Yaskawa INFORM job: sMulti_Axis_right_toolchange.JBI

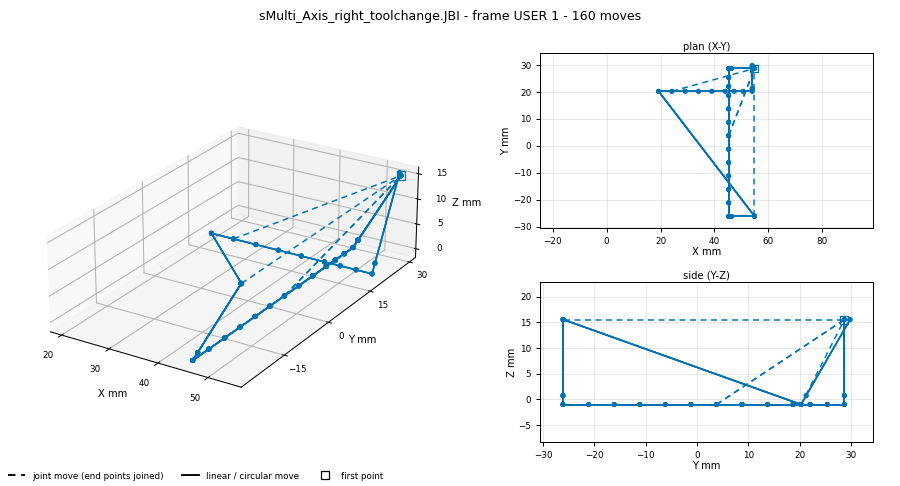
[picture p0: tool path of sMulti_Axis_right_toolchange.JBI in frame USER 1, 160 of 160 moves have a stored position in this frame; points joined in program order, loops and branches not executed]
/JOB
//NAME sMulti_Axis_right_toolchange
//POS
///NPOS 17,0,0,0,0,0
///USER 1
///TOOL 2
///POSTYPE USER
///RECTAN
///RCONF 1,0,0,0,0,0
C00000=50.999,-29.823,15.536,-90.000,-150.794,-116.565
C00001=50.999,-21.274,0.729,-90.000,-150.794,-116.565
C00002=50.999,-20.274,-1.003,-90.000,-150.794,-116.565
C00003=47.666,-20.274,-1.003,-90.000,-150.794,-116.565
C00004=44.332,-20.274,-1.003,-90.000,-150.794,-116.565
C00005=40.999,-20.274,-1.003,-90.000,-150.794,-116.565
C00006=36.223,-20.274,-1.003,-90.000,-150.794,-116.565
C00007=31.447,-20.274,-1.003,-90.000,-150.794,-116.565
C00008=26.671,-20.274,-1.003,-90.000,-150.794,-116.565
C00009=21.896,-20.274,-1.003,-90.000,-150.794,-116.565
C00010=17.120,-20.274,-1.003,-90.000,-150.794,-116.565
C00011=12.344,-20.274,-1.003,-90.000,-150.794,-116.565
C00012=7.568,-20.274,-1.003,-90.000,-150.794,-116.565
C00013=2.792,-20.274,-1.003,-90.000,-150.794,-116.565
C00014=-1.983,-20.274,-1.003,-90.000,-150.794,-116.565
C00015=-6.759,-20.274,-1.003,-90.000,-150.794,-116.565
C00016=-11.535,-20.274,-1.003,-90.000,-150.794,-116.565
C00017=-16.311,-20.274,-1.003,-90.000,-150.794,-116.565
C00018=-21.087,-20.274,-1.003,-90.000,-150.794,-116.565
C00019=-25.862,-20.274,-1.003,-90.000,-150.794,-116.565
C00020=-30.638,-20.274,-1.003,-90.000,-150.794,-116.565
C00021=-35.414,-20.274,-1.003,-90.000,-150.794,-116.565
C00022=-40.190,-20.274,-1.003,-90.000,-150.794,-116.565
C00023=-44.966,-20.274,-1.003,-90.000,-150.794,-116.565
C00024=-48.299,-20.274,-1.003,-90.000,-150.794,-116.565
C00025=-51.632,-20.274,-1.003,-90.000,-150.794,-116.565
C00026=-54.966,-20.274,-1.003,-90.000,-150.794,-116.565
C00027=-54.966,-21.274,0.729,-90.000,-150.794,-116.565
C00028=-54.966,-29.823,15.536,-90.000,-150.794,-116.565
C00000=53.984,-29.817,15.539,-90.000,-150.794,-116.565
C00001=53.984,-24.817,6.879,-90.000,-150.794,-116.565
C00002=53.984,-20.744,-0.175,-90.000,-150.794,-116.565
C00003=53.705,-20.407,-0.758,-90.000,-150.794,-116.565
C00004=53.031,-20.268,-1.000,-90.000,-150.794,-116.565
C00005=-55.536,-20.268,-1.000,-90.000,-150.794,-116.565
C00006=-56.209,-20.407,-0.758,-90.000,-150.794,-116.565
C00007=-56.488,-20.744,-0.175,-90.000,-150.794,-116.565
C00008=-56.488,-29.817,15.539,-90.000,-150.794,-116.565
C00000=-54.823,-30.003,15.536,180.000,-152.507,146.310
C00001=-46.274,-30.003,0.729,180.000,-152.507,146.310
C00002=-45.274,-30.003,-1.003,180.000,-152.507,146.310
C00003=-45.274,-26.669,-1.003,180.000,-152.507,146.310
C00004=-45.274,-23.336,-1.003,180.000,-152.507,146.310
C00005=-45.274,-20.003,-1.003,180.000,-152.507,146.310
C00006=-45.274,-15.558,-1.003,180.000,-152.507,146.310
C00007=-45.274,-11.113,-1.003,180.000,-152.507,146.310
C00008=-45.274,-6.668,-1.003,180.000,-152.507,146.310
C00009=-45.274,-2.223,-1.003,180.000,-152.507,146.310
C00010=-45.274,2.223,-1.003,180.000,-152.507,146.310
C00011=-45.274,6.668,-1.003,180.000,-152.507,146.310
C00012=-45.274,11.113,-1.003,180.000,-152.507,146.310
C00013=-45.274,15.558,-1.003,180.000,-152.507,146.310
C00014=-45.274,20.003,-1.003,-180.000,-152.507,146.310
C00015=-45.274,23.336,-1.003,-180.000,-152.507,146.310
C00016=-45.274,26.669,-1.003,-180.000,-152.507,146.310
C00017=-45.274,30.003,-1.003,-180.000,-152.507,146.310
C00018=-46.274,30.003,0.729,-180.000,-152.507,146.310
C00019=-54.823,30.003,15.536,-180.000,-152.507,146.310
C00000=54.301,-29.817,15.539,-90.000,-150.794,-116.565
C00001=54.301,-24.817,6.879,-90.000,-150.794,-116.565
C00002=54.301,-20.903,0.100,-90.000,-150.794,-116.565
C00003=53.929,-20.454,-0.678,-90.000,-150.794,-116.565
C00004=53.031,-20.268,-1.000,-90.000,-150.794,-116.565
C00005=-55.536,-20.268,-1.000,-90.000,-150.794,-116.565
C00006=-56.434,-20.454,-0.678,-90.000,-150.794,-116.565
C00007=-56.806,-20.903,0.100,-90.000,-150.794,-116.565
C00008=-56.806,-29.817,15.539,-90.000,-150.794,-116.565
C00000=-54.969,29.823,15.536,90.000,-150.794,63.435
C00001=-54.969,21.274,0.729,90.000,-150.794,63.435
C00002=-54.969,20.274,-1.003,90.000,-150.794,63.435
C00003=-51.636,20.274,-1.003,90.000,-150.794,63.435
C00004=-48.303,20.274,-1.003,90.000,-150.794,63.435
C00005=-44.969,20.274,-1.003,90.000,-150.794,63.435
C00006=-40.029,20.274,-1.003,90.000,-150.794,63.435
C00007=-35.088,20.274,-1.003,90.000,-150.794,63.435
C00008=-30.147,20.274,-1.003,90.000,-150.794,63.435
C00009=-25.206,20.274,-1.003,90.000,-150.794,63.435
C00010=-20.266,20.274,-1.003,90.000,-150.794,63.435
C00011=-15.325,20.274,-1.003,90.000,-150.794,63.435
C00012=-10.384,20.274,-1.003,90.000,-150.794,63.435
C00013=-5.443,20.274,-1.003,90.000,-150.794,63.435
C00014=-0.502,20.274,-1.003,90.000,-150.794,63.435
C00015=4.438,20.274,-1.003,90.000,-150.794,63.435
C00016=9.379,20.274,-1.003,90.000,-150.794,63.435
C00017=14.320,20.274,-1.003,90.000,-150.794,63.435
C00018=19.261,20.274,-1.003,90.000,-150.794,63.435
C00019=24.201,20.274,-1.003,90.000,-150.794,63.435
C00020=29.142,20.274,-1.003,90.000,-150.794,63.435
C00021=34.083,20.274,-1.003,90.000,-150.794,63.435
C00022=39.024,20.274,-1.003,90.000,-150.794,63.435
C00023=43.965,20.274,-1.003,90.000,-150.794,63.435
C00024=47.298,20.274,-1.003,90.000,-150.794,63.435
C00025=50.631,20.274,-1.003,90.000,-150.794,63.435
C00026=53.965,20.274,-1.003,90.000,-150.794,63.435
C00027=53.965,21.274,0.729,90.000,-150.794,63.435
C00028=53.965,29.823,15.536,90.000,-150.794,63.435
C00000=-54.969,29.823,15.536,90.000,-150.794,63.435
C00001=-54.969,21.274,0.729,90.000,-150.794,63.435
C00002=-54.969,20.274,-1.003,90.000,-150.794,63.435
C00003=-51.636,20.274,-1.003,90.000,-150.794,63.435
C00004=-48.303,20.274,-1.003,90.000,-150.794,63.435
C00005=-44.969,20.274,-1.003,90.000,-150.794,63.435
C00006=-40.029,20.274,-1.003,90.000,-150.794,63.435
C00007=-35.088,20.274,-1.003,90.000,-150.794,63.435
C00008=-30.147,20.274,-1.003,90.000,-150.794,63.435
C00009=-25.206,20.274,-1.003,90.000,-150.794,63.435
C00010=-20.266,20.274,-1.003,90.000,-150.794,63.435
C00011=-15.325,20.274,-1.003,90.000,-150.794,63.435
C00012=-10.384,20.274,-1.003,90.000,-150.794,63.435
C00013=-5.443,20.274,-1.003,90.000,-150.794,63.435
C00014=-0.502,20.274,-1.003,90.000,-150.794,63.435
C00015=4.438,20.274,-1.003,90.000,-150.794,63.435
C00016=9.379,20.274,-1.003,90.000,-150.794,63.435
C00017=14.320,20.274,-1.003,90.000,-150.794,63.435
C00018=19.261,20.274,-1.003,90.000,-150.794,63.435
C00019=24.201,20.274,-1.003,90.000,-150.794,63.435
C00020=29.142,20.274,-1.003,90.000,-150.794,63.435
C00021=34.083,20.274,-1.003,90.000,-150.794,63.435
C00022=39.024,20.274,-1.003,90.000,-150.794,63.435
C00023=43.965,20.274,-1.003,90.000,-150.794,63.435
C00024=47.298,20.274,-1.003,90.000,-150.794,63.435
C00025=50.631,20.274,-1.003,90.000,-150.794,63.435
C00026=53.965,20.274,-1.003,90.000,-150.794,63.435
C00027=53.965,21.274,0.729,90.000,-150.794,63.435
C00028=53.965,29.823,15.536,90.000,-150.794,63.435
C00000=54.817,28.503,15.539,0.000,-152.507,-33.690
C00001=46.268,28.503,0.732,0.000,-152.507,-33.690
C00002=45.268,28.503,-1.000,0.000,-152.507,-33.690
C00003=45.268,25.169,-1.000,0.000,-152.507,-33.690
C00004=45.268,21.836,-1.000,0.000,-152.507,-33.690
C00005=45.268,18.503,-1.000,0.000,-152.507,-33.690
C00006=45.268,13.573,-1.000,0.000,-152.507,-33.690
C00007=45.268,8.644,-1.000,0.000,-152.507,-33.690
C00008=45.268,3.715,-1.000,0.000,-152.507,-33.690
C00009=45.268,-1.214,-1.000,0.000,-152.507,-33.690
C00010=45.268,-6.144,-1.000,0.000,-152.507,-33.690
C00011=45.268,-11.073,-1.000,0.000,-152.507,-33.690
C00012=45.268,-16.002,-1.000,0.000,-152.507,-33.690
C00013=45.268,-19.336,-1.000,0.000,-152.507,-33.690
C00014=45.268,-22.669,-1.000,0.000,-152.507,-33.690
C00015=45.268,-26.002,-1.000,0.000,-152.507,-33.690
C00016=46.268,-26.002,0.732,0.000,-152.507,-33.690
C00017=54.817,-26.002,15.539,0.000,-152.507,-33.690
C00000=54.817,28.728,15.539,0.000,-152.507,-33.690
C00001=46.268,28.728,0.732,0.000,-152.507,-33.690
C00002=45.268,28.728,-1.000,0.000,-152.507,-33.690
C00003=45.268,25.395,-1.000,0.000,-152.507,-33.690
C00004=45.268,22.062,-1.000,0.000,-152.507,-33.690
C00005=45.268,18.728,-1.000,0.000,-152.507,-33.690
C00006=45.268,13.751,-1.000,0.000,-152.507,-33.690
C00007=45.268,8.773,-1.000,0.000,-152.507,-33.690
C00008=45.268,3.795,-1.000,0.000,-152.507,-33.690
C00009=45.268,-1.182,-1.000,0.000,-152.507,-33.690
C00010=45.268,-6.160,-1.000,0.000,-152.507,-33.690
C00011=45.268,-11.138,-1.000,0.000,-152.507,-33.690
C00012=45.268,-16.115,-1.000,0.000,-152.507,-33.690
C00013=45.268,-21.115,-1.000,0.000,-152.507,-33.690
C00014=45.268,-26.115,-1.000,0.000,-152.507,-33.690
C00015=46.268,-26.115,0.732,0.000,-152.507,-33.690
C00016=54.817,-26.115,15.539,0.000,-152.507,-33.690
//INST
///ATTR SC,RW,RJ
////FRAME USER 1
///GROUP1 RB1
///LVARS 2,0,0,0,0,0,0,0
NOP
SET LB000 1
SET LB001 25
MOVJ C00000 VJ=17
MOVL C00001 V=17 PL=LB000 ACC=LB001 DEC=LB001
' Lead In Move Starts
MOVL C00002 V=17 PL=LB000 ACC=LB001 DEC=LB001
' Cutting Move Starts
MOVL C00003 V=17 PL=LB000 ACC=LB001 DEC=LB001
MOVL C00004 V=17 PL=LB000 ACC=LB001 DEC=LB001
MOVL C00005 V=17 PL=LB000 ACC=LB001 DEC=LB001
MOVL C00006 V=17 PL=LB000 ACC=LB001 DEC=LB001
MOVL C00007 V=17 PL=LB000 ACC=LB001 DEC=LB001
MOVL C00008 V=17 PL=LB000 ACC=LB001 DEC=LB001
MOVL C00009 V=17 PL=LB000 ACC=LB001 DEC=LB001
MOVL C00010 V=17 PL=LB000 ACC=LB001 DEC=LB001
MOVL C00011 V=17 PL=LB000 ACC=LB001 DEC=LB001
MOVL C00012 V=17 PL=LB000 ACC=LB001 DEC=LB001
MOVL C00013 V=17 PL=LB000 ACC=LB001 DEC=LB001
MOVL C00014 V=17 PL=LB000 ACC=LB001 DEC=LB001
MOVL C00015 V=17 PL=LB000 ACC=LB001 DEC=LB001
MOVL C00016 V=17 PL=LB000 ACC=LB001 DEC=LB001
MOVL C00017 V=17 PL=LB000 ACC=LB001 DEC=LB001
MOVL C00018 V=17 PL=LB000 ACC=LB001 DEC=LB001
MOVL C00019 V=17 PL=LB000 ACC=LB001 DEC=LB001
MOVL C00020 V=17 PL=LB000 ACC=LB001 DEC=LB001
MOVL C00021 V=17 PL=LB000 ACC=LB001 DEC=LB001
MOVL C00022 V=17 PL=LB000 ACC=LB001 DEC=LB001
MOVL C00023 V=17 PL=LB000 ACC=LB001 DEC=LB001
MOVL C00024 V=17 PL=LB000 ACC=LB001 DEC=LB001
MOVL C00025 V=17 PL=LB000 ACC=LB001 DEC=LB001
MOVL C00026 V=17 PL=LB000 ACC=LB001 DEC=LB001
' Lead Out Move Starts
MOVL C00027 V=17 PL=LB000 ACC=LB001 DEC=LB001
' Rapid Move Starts
MOVL C00028 V=17 PL=LB000 ACC=LB001 DEC=LB001
' By Autodesk Fusion CAM 2.0.20494
' Tool = 8
' Spindle = 6000 RPM
' Set Position Level
' Set Acceleration
' Program Start
' First Toolpath Point
' Last Toolpath Point
MOVJ C00000 VJ=17
MOVL C00001 V=17 PL=LB000 ACC=LB001 DEC=LB001
' Plunge Move Starts
MOVL C00002 V=8 PL=LB000 ACC=LB001 DEC=LB001
' Lead In Move Starts
MOVL C00003 V=17 PL=LB000 ACC=LB001 DEC=LB001
MOVL C00004 V=17 PL=LB000 ACC=LB001 DEC=LB001
' Cutting Move Starts
MOVL C00005 V=17 PL=LB000 ACC=LB001 DEC=LB001
' Lead Out Move Starts
MOVL C00006 V=17 PL=LB000 ACC=LB001 DEC=LB001
MOVL C00007 V=17 PL=LB000 ACC=LB001 DEC=LB001
' Rapid Move Starts
MOVL C00008 V=17 PL=LB000 ACC=LB001 DEC=LB001
' By Autodesk Fusion CAM 2.0.20494
' Tool = 2
' Spindle = 5000 RPM
' Set Position Level
' Set Acceleration
' Program Start
' First Toolpath Point
' Last Toolpath Point
MOVJ C00000 VJ=17
MOVL C00001 V=17 PL=LB000 ACC=LB001 DEC=LB001
' Lead In Move Starts
MOVL C00002 V=17 PL=LB000 ACC=LB001 DEC=LB001
' Cutting Move Starts
MOVL C00003 V=17 PL=LB000 ACC=LB001 DEC=LB001
MOVL C00004 V=17 PL=LB000 ACC=LB001 DEC=LB001
MOVL C00005 V=17 PL=LB000 ACC=LB001 DEC=LB001
MOVL C00006 V=17 PL=LB000 ACC=LB001 DEC=LB001
MOVL C00007 V=17 PL=LB000 ACC=LB001 DEC=LB001
MOVL C00008 V=17 PL=LB000 ACC=LB001 DEC=LB001
MOVL C00009 V=17 PL=LB000 ACC=LB001 DEC=LB001
MOVL C00010 V=17 PL=LB000 ACC=LB001 DEC=LB001
MOVL C00011 V=17 PL=LB000 ACC=LB001 DEC=LB001
MOVL C00012 V=17 PL=LB000 ACC=LB001 DEC=LB001
MOVL C00013 V=17 PL=LB000 ACC=LB001 DEC=LB001
MOVL C00014 V=17 PL=LB000 ACC=LB001 DEC=LB001
MOVL C00015 V=17 PL=LB000 ACC=LB001 DEC=LB001
MOVL C00016 V=17 PL=LB000 ACC=LB001 DEC=LB001
MOVL C00017 V=17 PL=LB000 ACC=LB001 DEC=LB001
' Lead Out Move Starts
MOVL C00018 V=17 PL=LB000 ACC=LB001 DEC=LB001
' Rapid Move Starts
MOVL C00019 V=17 PL=LB000 ACC=LB001 DEC=LB001
' By Autodesk Fusion CAM 2.0.20494
' Tool = 8
' Spindle = 6000 RPM
' Set Position Level
' Set Acceleration
' Program Start
' First Toolpath Point
' Last Toolpath Point
MOVJ C00000 VJ=17
MOVL C00001 V=17 PL=LB000 ACC=LB001 DEC=LB001
' Plunge Move Starts
MOVL C00002 V=8 PL=LB000 ACC=LB001 DEC=LB001
' Lead In Move Starts
MOVL C00003 V=17 PL=LB000 ACC=LB001 DEC=LB001
MOVL C00004 V=17 PL=LB000 ACC=LB001 DEC=LB001
' Cutting Move Starts
MOVL C00005 V=17 PL=LB000 ACC=LB001 DEC=LB001
' Lead Out Move Starts
MOVL C00006 V=17 PL=LB000 ACC=LB001 DEC=LB001
MOVL C00007 V=17 PL=LB000 ACC=LB001 DEC=LB001
' Rapid Move Starts
MOVL C00008 V=17 PL=LB000 ACC=LB001 DEC=LB001
' By Autodesk Fusion CAM 2.0.20494
' Tool = 8
' Spindle = 6000 RPM
' Set Position Level
' Set Acceleration
' Program Start
' First Toolpath Point
' Last Toolpath Point
MOVJ C00000 VJ=17
MOVL C00001 V=17 PL=LB000 ACC=LB001 DEC=LB001
' Lead In Move Starts
MOVL C00002 V=17 PL=LB000 ACC=LB001 DEC=LB001
' Cutting Move Starts
MOVL C00003 V=17 PL=LB000 ACC=LB001 DEC=LB001
MOVL C00004 V=17 PL=LB000 ACC=LB001 DEC=LB001
MOVL C00005 V=17 PL=LB000 ACC=LB001 DEC=LB001
MOVL C00006 V=17 PL=LB000 ACC=LB001 DEC=LB001
MOVL C00007 V=17 PL=LB000 ACC=LB001 DEC=LB001
MOVL C00008 V=17 PL=LB000 ACC=LB001 DEC=LB001
MOVL C00009 V=17 PL=LB000 ACC=LB001 DEC=LB001
MOVL C00010 V=17 PL=LB000 ACC=LB001 DEC=LB001
MOVL C00011 V=17 PL=LB000 ACC=LB001 DEC=LB001
MOVL C00012 V=17 PL=LB000 ACC=LB001 DEC=LB001
MOVL C00013 V=17 PL=LB000 ACC=LB001 DEC=LB001
MOVL C00014 V=17 PL=LB000 ACC=LB001 DEC=LB001
MOVL C00015 V=17 PL=LB000 ACC=LB001 DEC=LB001
MOVL C00016 V=17 PL=LB000 ACC=LB001 DEC=LB001
MOVL C00017 V=17 PL=LB000 ACC=LB001 DEC=LB001
MOVL C00018 V=17 PL=LB000 ACC=LB001 DEC=LB001
MOVL C00019 V=17 PL=LB000 ACC=LB001 DEC=LB001
MOVL C00020 V=17 PL=LB000 ACC=LB001 DEC=LB001
MOVL C00021 V=17 PL=LB000 ACC=LB001 DEC=LB001
MOVL C00022 V=17 PL=LB000 ACC=LB001 DEC=LB001
MOVL C00023 V=17 PL=LB000 ACC=LB001 DEC=LB001
MOVL C00024 V=17 PL=LB000 ACC=LB001 DEC=LB001
MOVL C00025 V=17 PL=LB000 ACC=LB001 DEC=LB001
MOVL C00026 V=17 PL=LB000 ACC=LB001 DEC=LB001
' Lead Out Move Starts
MOVL C00027 V=17 PL=LB000 ACC=LB001 DEC=LB001
' Rapid Move Starts
MOVL C00028 V=17 PL=LB000 ACC=LB001 DEC=LB001
' By Autodesk Fusion CAM 2.0.20494
' Tool = 8
' Spindle = 6000 RPM
' Set Position Level
' Set Acceleration
' Program Start
' First Toolpath Point
' Last Toolpath Point
MOVJ C00000 VJ=17
MOVL C00001 V=17 PL=LB000 ACC=LB001 DEC=LB001
' Lead In Move Starts
MOVL C00002 V=17 PL=LB000 ACC=LB001 DEC=LB001
' Cutting Move Starts
MOVL C00003 V=17 PL=LB000 ACC=LB001 DEC=LB001
MOVL C00004 V=17 PL=LB000 ACC=LB001 DEC=LB001
MOVL C00005 V=17 PL=LB000 ACC=LB001 DEC=LB001
MOVL C00006 V=17 PL=LB000 ACC=LB001 DEC=LB001
MOVL C00007 V=17 PL=LB000 ACC=LB001 DEC=LB001
MOVL C00008 V=17 PL=LB000 ACC=LB001 DEC=LB001
MOVL C00009 V=17 PL=LB000 ACC=LB001 DEC=LB001
MOVL C00010 V=17 PL=LB000 ACC=LB001 DEC=LB001
MOVL C00011 V=17 PL=LB000 ACC=LB001 DEC=LB001
MOVL C00012 V=17 PL=LB000 ACC=LB001 DEC=LB001
MOVL C00013 V=17 PL=LB000 ACC=LB001 DEC=LB001
MOVL C00014 V=17 PL=LB000 ACC=LB001 DEC=LB001
MOVL C00015 V=17 PL=LB000 ACC=LB001 DEC=LB001
MOVL C00016 V=17 PL=LB000 ACC=LB001 DEC=LB001
MOVL C00017 V=17 PL=LB000 ACC=LB001 DEC=LB001
MOVL C00018 V=17 PL=LB000 ACC=LB001 DEC=LB001
MOVL C00019 V=17 PL=LB000 ACC=LB001 DEC=LB001
MOVL C00020 V=17 PL=LB000 ACC=LB001 DEC=LB001
MOVL C00021 V=17 PL=LB000 ACC=LB001 DEC=LB001
MOVL C00022 V=17 PL=LB000 ACC=LB001 DEC=LB001
MOVL C00023 V=17 PL=LB000 ACC=LB001 DEC=LB001
MOVL C00024 V=17 PL=LB000 ACC=LB001 DEC=LB001
MOVL C00025 V=17 PL=LB000 ACC=LB001 DEC=LB001
MOVL C00026 V=17 PL=LB000 ACC=LB001 DEC=LB001
' Lead Out Move Starts
MOVL C00027 V=17 PL=LB000 ACC=LB001 DEC=LB001
' Rapid Move Starts
MOVL C00028 V=17 PL=LB000 ACC=LB001 DEC=LB001
' By Autodesk Fusion CAM 2.0.20494
' Tool = 8
' Spindle = 6000 RPM
' Set Position Level
' Set Acceleration
' Program Start
' First Toolpath Point
' Last Toolpath Point
MOVJ C00000 VJ=17
MOVL C00001 V=17 PL=LB000 ACC=LB001 DEC=LB001
' Lead In Move Starts
MOVL C00002 V=17 PL=LB000 ACC=LB001 DEC=LB001
' Cutting Move Starts
MOVL C00003 V=17 PL=LB000 ACC=LB001 DEC=LB001
MOVL C00004 V=17 PL=LB000 ACC=LB001 DEC=LB001
MOVL C00005 V=17 PL=LB000 ACC=LB001 DEC=LB001
MOVL C00006 V=17 PL=LB000 ACC=LB001 DEC=LB001
MOVL C00007 V=17 PL=LB000 ACC=LB001 DEC=LB001
MOVL C00008 V=17 PL=LB000 ACC=LB001 DEC=LB001
MOVL C00009 V=17 PL=LB000 ACC=LB001 DEC=LB001
MOVL C00010 V=17 PL=LB000 ACC=LB001 DEC=LB001
MOVL C00011 V=17 PL=LB000 ACC=LB001 DEC=LB001
MOVL C00012 V=17 PL=LB000 ACC=LB001 DEC=LB001
MOVL C00013 V=17 PL=LB000 ACC=LB001 DEC=LB001
MOVL C00014 V=17 PL=LB000 ACC=LB001 DEC=LB001
MOVL C00015 V=17 PL=LB000 ACC=LB001 DEC=LB001
' Lead Out Move Starts
MOVL C00016 V=17 PL=LB000 ACC=LB001 DEC=LB001
' Rapid Move Starts
MOVL C00017 V=17 PL=LB000 ACC=LB001 DEC=LB001
' By Autodesk Fusion CAM 2.0.20494
' Tool = 8
' Spindle = 6000 RPM
' Set Position Level
' Set Acceleration
' Program Start
' First Toolpath Point
' Last Toolpath Point
MOVJ C00000 VJ=17
MOVL C00001 V=17 PL=LB000 ACC=LB001 DEC=LB001
' Lead In Move Starts
MOVL C00002 V=17 PL=LB000 ACC=LB001 DEC=LB001
' Cutting Move Starts
MOVL C00003 V=17 PL=LB000 ACC=LB001 DEC=LB001
MOVL C00004 V=17 PL=LB000 ACC=LB001 DEC=LB001
MOVL C00005 V=17 PL=LB000 ACC=LB001 DEC=LB001
MOVL C00006 V=17 PL=LB000 ACC=LB001 DEC=LB001
MOVL C00007 V=17 PL=LB000 ACC=LB001 DEC=LB001
MOVL C00008 V=17 PL=LB000 ACC=LB001 DEC=LB001
MOVL C00009 V=17 PL=LB000 ACC=LB001 DEC=LB001
MOVL C00010 V=17 PL=LB000 ACC=LB001 DEC=LB001
MOVL C00011 V=17 PL=LB000 ACC=LB001 DEC=LB001
MOVL C00012 V=17 PL=LB000 ACC=LB001 DEC=LB001
MOVL C00013 V=17 PL=LB000 ACC=LB001 DEC=LB001
MOVL C00014 V=17 PL=LB000 ACC=LB001 DEC=LB001
' Lead Out Move Starts
MOVL C00015 V=17 PL=LB000 ACC=LB001 DEC=LB001
' Rapid Move Starts
MOVL C00016 V=17 PL=LB000 ACC=LB001 DEC=LB001
' By Autodesk Fusion CAM 2.0.20494
' Tool = 2
' Spindle = 5000 RPM
' Set Position Level
' Set Acceleration
' Program Start
' First Toolpath Point
END
